Staubli VAL3: iFluorOpen.pgx

public program iFluorOpen(num& nNum[] (dimensions=1))
begin
  nNum=dioGet(iFluorOpen)
end
